FUNCTION_BLOCK E_TABLE_CTRL (* Support function block for E_TABLE *)
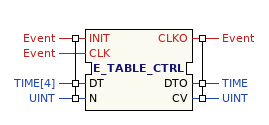
  EVENT_INPUT
    INIT WITH DT, N;
    CLK;
  END_EVENT
  EVENT_OUTPUT
    CLKO WITH DTO, CV;
  END_EVENT
  VAR_INPUT
    DT : ARRAY [0..3] OF TIME;
    N : UINT; (* Actual number of time steps *)
  END_VAR
  VAR_OUTPUT
    DTO : TIME; (* Current delay interval *)
    CV : UINT; (* Current event index, 0..N-1 *)
  END_VAR
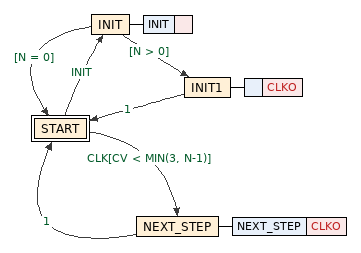
  EC_STATES
    START; (* Initial State *)
    INIT : INIT;
    INIT1 : -> CLKO;
    NEXT_STEP : NEXT_STEP -> CLKO;
  END_STATES
  EC_TRANSITIONS
    START TO INIT := INIT;
    INIT TO START := [N = 0];
    INIT TO INIT1 := [N > 0];
    INIT1 TO START := 1;
    START TO NEXT_STEP := CLK[CV < MIN(3, N-1)];
    NEXT_STEP TO START := 1;
  END_TRANSITIONS
  ALGORITHM INIT IN ST:
CV := 0;
DTO := DT[0];
  END_ALGORITHM
  ALGORITHM NEXT_STEP IN ST:
CV := CV +1;
DTO := DT[CV];
  END_ALGORITHM
END_FUNCTION_BLOCK
